FUNCTION_BLOCK diag_j
VAR_INPUT
	v: ARRAY[0..10] OF LREAL;
END_VAR
VAR_OUTPUT
	b_d: ARRAY[0..120] OF LREAL;
END_VAR
VAR
	j: DINT;
END_VAR



FOR j := 0 TO 120 DO 
    b_d[j] := 0.0;
END_FOR;


FOR j := 0 TO 10 DO 
    b_d[j + (11 * j)] := v[j];
END_FOR;

END_FUNCTION_BLOCK

(* stored: Version 1.1.0.1, ProductVersion 3.1.4022.7
   POU diag_j: Id {25f895e2-7feb-4dec-975a-45d0c0616ce7}, SpecialFunc None *)
